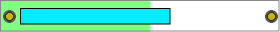
VISUALIZATION CylSimul  // 280x32
VAR_IN_OUT
	currPosPercent:LREAL;
	sensorFwd: BOOL;
	sensorBwd: BOOL;
END_VAR
    Rectangle (0,0 150x32)
    Rectangle (20,8 150x16)
        p3528305787: currPosPercent
        p874137650: currPosPercent
    Lamp1 (2,9 15x15), variable: sensorBwd, style: Lamp-Lamp1-Yellow
    Lamp1 (264,9 15x15), variable: sensorFwd, style: Lamp-Lamp1-Yellow
END_VISUALIZATION

(* stored: Version 1.1.0.1, ProductVersion 3.1.4024.12
   Visu CylSimul: Id {81012372-df1f-4ca1-b029-2696a81b1672} *)
